# EPICS StreamDevice protocol: AFG3XXXSup/devAFG3XXX.proto
InTerminator = '\n';
#ReplyTimeout = 2000;

getIDN {
    out "*IDN?";
    #Read no more that 39 chars (EPICS limit)
    in "%/(.{0,39})/";
    ExtraInput = Ignore;
}

getStatus {
    out "OUTP\$1:STAT?";
    in "%d";
    ExtraInput = Ignore;
}

setStatus {
    out "OUTP\$1:STAT %d";
}

getFunction {
    out "SOUR\$1:FUNC:SHAP?";
    in "%{SIN|SQU|PULS|RAMP|PRN|DC|SINC|GAUS|LOR|ERIS|EDEC|HAV}";
    ExtraInput = Ignore;
}

setFunction {
    out "SOUR\$1:FUNC:SHAP %{SIN|SQU|PULS|RAMP|PRN|DC|SINC|GAUS|LOR|ERIS|EDEC|HAV}";
}

getImpedance {
    out "OUTP\$1:IMP?";
    in "%f";
    ExtraInput = Ignore;
}

setImpedance {
    out "OUTP\$1:IMP %s";
}

getPolarity {
    out "OUTP\$1:POL?";
    in "%{NORM|INV}";
    ExtraInput = Ignore;
}

setPolarity {
    out "OUTP\$1:POL %{NORM|INV}";
}

getVoltage {
    out "SOUR\$1:VOLT?";
    in "%f";
    ExtraInput = Ignore;
}

setVoltage {
    out "SOUR\$1:VOLT %s";
}

getVoltageUnits {
    out "SOUR\$1:VOLT:UNIT?";
    in "%{VPP|VRMS|DBM}";
    ExtraInput = Ignore;
}

setVoltageUnits {
    out "SOUR\$1:VOLT:UNIT %{VPP|VRMS|DBM}";
}

getVoltageLowLimit {
    out "SOUR\$1:VOLT:LIM:LOW?";
    in "%f";
    ExtraInput = Ignore;
}

setVoltageLowLimit {
    out "SOUR\$1:VOLT:LIM:LOW %s";
}

getVoltageHighLimit {
    out "SOUR\$1:VOLT:LIM:HIGH?";
    in "%f";
    ExtraInput = Ignore;
}

setVoltageHighLimit {
    out "SOUR\$1:VOLT:LIM:HIGH %s";
}

getVoltageLowLevel {
    out "SOUR\$1:VOLT:LEV:IMM:LOW?";
    in "%f";
    ExtraInput = Ignore;
}

setVoltageLowLevel {
    out "SOUR\$1:VOLT:LEV:IMM:LOW %s";
}

getVoltageHighLevel {
    out "SOUR\$1:VOLT:LEV:IMM:HIGH?";
    in "%f";
    ExtraInput = Ignore;
}

setVoltageHighLevel {
    out "SOUR\$1:VOLT:LEV:IMM:HIGH %s";
}

getVoltageOffset {
    out "SOUR\$1:VOLT:LEV:IMM:OFFS?";
    in "%f";
    ExtraInput = Ignore;
}

setVoltageOffset {
    out "SOUR\$1:VOLT:LEV:IMM:OFFS %s";
}

getFrequency {
    out "SOUR\$1:FREQ:FIX?";
    in "%f";
    ExtraInput = Ignore;
}

setFrequency {
    out "SOUR\$1:FREQ:FIX %s";
}

getPhase {
    out "SOUR\$1:PHASE:ADJ?";
    in "%f";
    ExtraInput = Ignore;
}

setPhase {
    out "SOUR\$1:PHASE:ADJ %s";
}

getBurstStatus {
    out "SOUR\$1:BURS:STAT?";
    in "%d";
    ExtraInput = Ignore;
}

setBurstStatus {
    out "SOUR\$1:BURS:STAT %{ON|OFF}";
}

getBurstMode {
    out "SOUR\$1:BURS:MODE?";
    in "%{TRIG|GAT}";
    ExtraInput = Ignore;
}

setBurstMode {
    out "SOUR\$1:BURS:MODE %{TRIG|GAT}";
}

getBurstNCycles {
    out "SOUR\$1:BURS:NCYC?";
    in "%f";
    ExtraInput = Ignore;
}

setBurstNCycles {
    out "SOUR\$1:BURS:NCYC %s";
}

getBurstTimeDelay {
    out "SOUR\$1:BURS:TDEL?";
    in "%f";
    ExtraInput = Ignore;
}

setBurstTimeDelay {
    out "SOUR\$1:BURS:TDEL %s";
}

getFrequencyMode {
    out "SOUR\$1:FREQ:MODE?";
    in "%{CW|FIX|SWE}";
    ExtraInput = Ignore;
}

setFrequencyMode {
    out "SOUR\$1:FREQ:MODE %{CW|FIX|SWE}";
}

getSweepSpan {
    out "SOUR\$1:FREQ:SPAN?";
    in "%f";
    ExtraInput = Ignore;
}

setSweepSpan {
    out "SOUR\$1:FREQ:SPAN %s";
}

getSweepStart {
    out "SOUR\$1:FREQ:STAR?";
    in "%f";
    ExtraInput = Ignore;
}

setSweepStart {
    out "SOUR\$1:FREQ:STAR %s";
}

getSweepStop {
    out "SOUR\$1:FREQ:STOP?";
    in "%f";
    ExtraInput = Ignore;
}

setSweepStop {
    out "SOUR\$1:FREQ:STOP %s";
}

getSweepHoldTime {
    out "SOUR\$1:SWE:HTIM?";
    in "%f";
    ExtraInput = Ignore;
}

setSweepHoldTime {
    out "SOUR\$1:SWE:HTIM %s";
}

getSweepMode {
    out "SOUR\$1:SWE:MODE?";
    in "%{AUTO|MAN}";
    ExtraInput = Ignore;
}

setSweepMode {
    out "SOUR\$1:SWE:MODE %{AUTO|MAN}";
}

getSweepReturnTime {
    out "SOUR\$1:SWE:RTIM?";
    in "%f";
    ExtraInput = Ignore;
}

setSweepReturnTime {
    out "SOUR\$1:SWE:RTIM %s";
}

getSweepSpacing {
    out "SOUR\$1:SWE:SPAC?";
    in "%s";
    ExtraInput = Ignore;
}

setSweepSpacing {
    out "SOUR\$1:SWE:SPAC %{LIN|LOG}";
}

getSweepTime {
    out "SOUR\$1:SWE:TIME?";
    in "%f";
    ExtraInput = Ignore;
}

setSweepTime {
    out "SOUR\$1:SWE:TIME %s";
}

trigger {
    out "*TRG";
}
